# EPICS autosave request: iocBoot/iocSolaris/auto_positions.req
$(P)SM1.OFF
$(P)SM1.DVAL
$(P)SM2.OFF
$(P)SM2.DVAL
$(P)SM3.OFF
$(P)SM3.DVAL
$(P)SM4.OFF
$(P)SM4.DVAL
$(P)SM5.OFF
$(P)SM5.DVAL
$(P)SM6.OFF
$(P)SM6.DVAL
$(P)SM7.OFF
$(P)SM7.DVAL
$(P)SM8.OFF
$(P)SM8.DVAL
